# EPICS autosave request: iocBoot/gmca_23i_ioc1/dbSave/BP_Hd3_.req
%
% BURT Request File
%
% $(P)BP:Kb:  BPM @ KB mirrors position
%
file assy.req ASSY=$(P)BP:Hd3
file mtr1.req MTR1=$(P)BP:mh3z
file drv1.req DRV1=$(P)BP:H3Z

$(P)BP:H3Z:RqsPosMem1
$(P)BP:H3Z:RqsPosMem2
$(P)BP:H3Z:RqsPosMem3
$(P)BP:H3Z:RqsPosMem4

$(P)BP:H3Z:RqsPosMem1.DESC
$(P)BP:H3Z:RqsPosMem2.DESC
$(P)BP:H3Z:RqsPosMem3.DESC
$(P)BP:H3Z:RqsPosMem4.DESC
